KUKA KRL program: Spindle.src

&ACCESS RV
DEF Spindle ( )

END

GLOBAL DEF SpindleInit ( )

   CONTINUE
   gDOSpindleEnable = TRUE

END

GLOBAL DEF SpindleRun (lrSpindleRPM :IN, FI_DIRECTION:IN)
   INT lrSpindleRPM
   DECL TYPMillDirection FI_DIRECTION

   CONTINUE

   gbRobControlActive = TRUE
   gDOSpindleEnable = TRUE
   WAIT FOR gDISpindleEnableOK == TRUE

   SWITCH FI_DIRECTION
      CASE #CLOCKWISE
         gISetSpeed = -lrSpindleRPM
         ;gbDirectionClockwise=TRUE
      CASE #COUNTERCLOCKWISE
         gISetSpeed = lrSpindleRPM
         ;gbDirectionClockwise=FALSE
   ENDSWITCH

END

GLOBAL DEF SpindleStop ( )

   gISetSpeed = 0
   ;;WAIT SEC 0

   gDOSpindleEnable = FALSE
   WAIT FOR gDISpindleEnableOK == FALSE
   gbRobControlActive = FALSE
END

GLOBAL DEF SpindleSetSpeed (lnSpeed :IN )
   INT lnSpeed

   gISetSpeed = lnSpeed

END
